// TIA Portal V20 export
// export: Created 2025-12-01T14:56:14.6294284Z, ExportSetting None, DisplayName Totally Integrated Automation Portal, DisplayVersion V20 Update 3, DisplayName TIA Portal Openness, DisplayVersion V20 Update 3, DisplayName TIA Portal Version Control Interface, DisplayVersion V20 Update 3, DisplayName STEP 7 Professional, DisplayVersion V20 Update 3, DisplayName STEP 7 Safety, DisplayVersion V20 Update 2, DisplayName WinCC Basic/Comfort/Advanced, DisplayVersion V20 Update 3, DisplayName WinCC Professional, DisplayVersion V20 Update 3, DisplayName WinCC Unified, DisplayVersion V20 Update 3
TYPE "ROUT_Conf_Bucle_Lect_SCR"
   STRUCT
      Modelo : UInt := 5;   // (0) DL PB (1) SICK PB (2) SICK_A PB (5) SICK PN (6) SICK_A PN
      AddresInicial : UInt := 0;   // Direccion Entrada / Salida del Primer Nodo de la Red
      NodoInicial : UInt := 0;   // Primer Nodo de la Red (ID profinet)
      NodoFinal : UInt := 0;   // Ultimo Nodo de la Red (ID profinet)
      Numero_Red : UInt := 1;   // Número de red en la que estan los scanners
      DB_NodosPresentes : UInt := 927;   // DD de Nodos Presentes en la Red
      SCR_Actual : UInt;   // Numero de SCR actual de la Red
   END_STRUCT;
END_TYPE
